(* IEC 61131-3 sources: TCPComm/src/Ar/TCPComm, 4 files *)

(* ---- TCPConnectionMgr.typ ---- *)
(*
 * File: TCPConnectionMgr.typ
 * Copyright (c) 2023 Loupe
 * https://loupe.team
 *
 * This file is part of TCPComm, licensed under the MIT License.
 *
 *)

TYPE
	TCPCOMM_MODE_enum :
		(
		TCPCOMM_MODE_SERVER := 50000,
		TCPCOMM_MODE_CLIENT
		);
	TCPCOMM_ERR_enum :
		(
		TCPCOMM_ERR_INVALIDINPUT := 50000,
		TCPCOMM_ERR_SENDDATATOOLARGE,
		TCPCOMM_ERR_
		);
	TCPCOMM_ST_enum :
		(
		TCPCOMM_ST_CLOSED,
		TCPCOMM_ST_OPENING,
		TCPCOMM_ST_IOCTL,
		TCPCOMM_ST_LISTEN,
		TCPCOMM_ST_RUNNING,
		TCPCOMM_ST_CLOSE_CONNECTION,
		TCPCOMM_ST_CLOSING,
		TCPCOMM_ST_ERROR
		);
	TCPCOMM_SEND_ST_enum :
		(
		TCPCOMM_SEND_ST_IDLE,
		TCPCOMM_SEND_ST_SEND
		);
	TCPCOMM_RECV_ST_enum :
		(
		TCPCOMM_RECV_ST_READ
		);
	TCPConnection_Desc_typ : 	STRUCT
		IPAddress : STRING[TCPCOMM_STRLEN_IPADDRESS];
		Port : UINT;
		Ident : UINT;
		UID : UDINT;
	END_STRUCT;
	TCPConnectionMgr_Int_FUB_typ : 	STRUCT
		Open : TcpOpen;
		OpenSSL : TcpOpenSsl;
		Ioctl : TcpIoctl;
		Server : TcpServer;
		Client : TcpClient;
		Close : TcpClose;
	END_STRUCT;
	TCPConnectionMgr_Internal_typ : 	STRUCT
		FUB : TCPConnectionMgr_Int_FUB_typ;
		CommState : TCPCOMM_ST_enum;
		Mode : TCPCOMM_MODE_enum;
		Ident : UDINT;
		ConnectionUID : UDINT;
	END_STRUCT;
	TCPConnectionMgr_OUT_typ : 	STRUCT
		NewConnectionAvailable : BOOL;
		Connection : TCPConnection_Desc_typ;
		Error : BOOL;
		ErrorID : UINT;
		ErrorString : STRING[TCPCOMM_STRLEN_ERRORSTRING];
	END_STRUCT;
	TCPConnectionMgr_IN_CFG_typ : 	STRUCT
		Mode : TCPCOMM_MODE_enum;
		LocalIPAddress : STRING[TCPCOMM_STRLEN_IPADDRESS];
		LocalPort : UINT;
		RemoteIPAddress : STRING[TCPCOMM_STRLEN_IPADDRESS];
		RemotePort : UINT;
		SendBufferSize : UDINT;
		UseSSL : BOOL;
		SSLCertificate : UDINT;
	END_STRUCT;
	TCPConnectionMgr_IN_CMD_typ : 	STRUCT
		Enable : BOOL;
		AcknowledgeConnection : BOOL;
		AcknowledgeError : BOOL;
	END_STRUCT;
	TCPConnectionMgr_IN_typ : 	STRUCT
		CMD : TCPConnectionMgr_IN_CMD_typ;
		CFG : TCPConnectionMgr_IN_CFG_typ;
	END_STRUCT;
	TCPConnectionMgr_typ : 	STRUCT
		IN : TCPConnectionMgr_IN_typ;
		OUT : TCPConnectionMgr_OUT_typ;
		Internal : TCPConnectionMgr_Internal_typ;
	END_STRUCT;
END_TYPE

(* ---- TCPStream.typ ---- *)
(*
 * File: TCPStream.typ
 * Copyright (c) 2023 Loupe
 * https://loupe.team
 *
 * This file is part of TCPComm, licensed under the MIT License.
 *
 *)

(*For each client lets instantiate an interface*)

TYPE
	TCPStream_Int_Debug_Mng_typ : 	STRUCT
		New_Member : {REDUND_UNREPLICABLE} USINT;
	END_STRUCT;
	TCPStream_Int_Debug_Recv_typ : 	STRUCT
		enable : {REDUND_UNREPLICABLE} ARRAY[0..1]OF BOOL;
		status : {REDUND_UNREPLICABLE} ARRAY[0..1]OF UINT;
	END_STRUCT;
	TCPStream_Int_Debug_Send_typ : 	STRUCT
		New_Member : {REDUND_UNREPLICABLE} USINT;
	END_STRUCT;
	TCPStream_Int_Debug_typ : 	STRUCT
		manage : {REDUND_UNREPLICABLE} TCPStream_Int_Debug_Mng_typ;
		receive : {REDUND_UNREPLICABLE} TCPStream_Int_Debug_Recv_typ;
		send : {REDUND_UNREPLICABLE} TCPStream_Int_Debug_Send_typ;
	END_STRUCT;
	TCPStream_Int_FUB_typ : 	STRUCT
		Send : TcpSend;
		Receive : TcpRecv;
		Close : TcpClose;
	END_STRUCT;
	TCPStream_Internal_typ : 	STRUCT
		CommState : TCPCOMM_ST_enum;
		Ident : UDINT;
		UID : UDINT;
		FUB : TCPStream_Int_FUB_typ;
		debug : {REDUND_UNREPLICABLE} TCPStream_Int_Debug_typ;
	END_STRUCT;
	TCPStream_OUT_typ : 	STRUCT
		Connection : TCPConnection_Desc_typ;
		Active : BOOL;
		Receiving : BOOL;
		DataReceived : BOOL;
		ReceivedDataLength : UDINT;
		Sending : BOOL;
		DataSent : BOOL;
		SentDataLength : UDINT;
		Error : BOOL;
		ErrorID : UINT;
		ErrorString : STRING[TCPCOMM_STRLEN_ERRORSTRING];
	END_STRUCT;
	TCPStream_IN_PAR_typ : 	STRUCT
		Connection : TCPConnection_Desc_typ;
		pReceiveData : UDINT;
		MaxReceiveLength : UDINT;
		ReceiveFlags : UINT;
		AllowContinuousReceive : BOOL;
		pSendData : UDINT;
		SendLength : UDINT;
		SendFlags : UINT;
		AllowContinuousSend : BOOL;
	END_STRUCT;
	TCPStream_IN_CMD_typ : 	STRUCT
		Receive : BOOL;
		Send : BOOL;
		Close : BOOL;
		AcknowledgeData : BOOL;
		AcknowledgeError : BOOL;
	END_STRUCT;
	TCPStream_IN_typ : 	STRUCT
		CMD : TCPStream_IN_CMD_typ;
		PAR : TCPStream_IN_PAR_typ;
	END_STRUCT;
	TCPStream_typ : 	STRUCT
		IN : TCPStream_IN_typ;
		OUT : TCPStream_OUT_typ;
		Internal : TCPStream_Internal_typ;
	END_STRUCT;
END_TYPE

(* ---- TCPComm.fun ---- *)
(*
 * File: TCPComm.fun
 * Copyright (c) 2023 Loupe
 * https://loupe.team
 *
 * This file is part of TCPComm, licensed under the MIT License.
 *
 *)

FUNCTION TCPManageConnection : UINT (*Cyclic function for managing TCP communications*) (*$GROUP=User*)
	VAR_IN_OUT
		t : TCPConnectionMgr_typ;
	END_VAR
END_FUNCTION

FUNCTION TCPStreamReceive : UINT (*Cyclic function to receive packets of data*) (*$GROUP=User*)
	VAR_IN_OUT
		t : TCPStream_typ;
	END_VAR
END_FUNCTION

FUNCTION TCPStreamSend : UINT (*Cyclic function to send packets of data*) (*$GROUP=User*)
	VAR_IN_OUT
		t : TCPStream_typ;
	END_VAR
END_FUNCTION

(* ---- TCPComm.var ---- *)
(*
 * File: TCPComm.var
 * Copyright (c) 2023 Loupe
 * https://loupe.team
 *
 * This file is part of TCPComm, licensed under the MIT License.
 *
 *)

VAR CONSTANT
	TCPCOMM_STRLEN_IPADDRESS : USINT := 255;
	TCPCOMM_STRLEN_ERRORSTRING : UINT := 320;
END_VAR
